{attribute 'qualified_only'}
{attribute 'strict'}
TYPE E_JANSSEN_STATUS :
(
	NOT_INIT	:= -1,
	IDLE		:= 0,
	ERROR		:= 1,
	BUSY		:= 2
);
END_TYPE

(* stored: Version 1.1.0.1, ProductVersion 3.1.4024.12
   DUT E_JANSSEN_STATUS: Id {ac32da46-a2a6-4d67-8514-ceb1d8e38cc4} *)
